# EPICS substitutions: siteApps/KoBRA_MAG-1-0/kobramagnetApp/Db/danfysik.substitutions
file "db/danfysikMps9700.template"
{
	pattern { device,			port,		inom,	imax,	imin,	ilim,	vnom,	vmax,	vmin }
		{ MEBT-QM3:Danfysik,	SYS9700,	350,	330,	-330,	25,		60,		60,		-60  }
}
